PROGRAM Main1ms
VAR
	mcModules		: ARRAY [1..mcGvl.cMaxModuleCapacity] OF FB_mcModuleBase;
	mcCount			: UINT;
END_VAR

A_mcCyclic();

ACTION A_mcCyclic:
mcGvl.OperationMode(); // Operation mode 
mcGvl.AxesConfigurator(); // Configurator to set number of axes
mcGvl.ModulesConfigurator(); // Configurator to set number of modules

FOR mcCount := 1 TO mcGvl.ModulesConfigurator.uiNoModulesActive DO
	mcModules[mcCount]();
END_FOR;
END_ACTION

END_PROGRAM

(* stored: Version 1.1.0.1, ProductVersion 3.1.4024.6
   POU Main1ms: Id {3580f847-e6d0-45a6-ba8f-b4c0385d5404}, SpecialFunc None
   Action A_mcCyclic: Id {4fd36bd2-0cdb-47c0-85db-8410bde7dda1} *)
